{attribute 'GeneratedUsingTerminal: KL9940-0050'}
{attribute addProperty BoxType "KL9940-0050"}
{attribute addProperty Id "Channel_1AT %I*Channel_954C2EED0"}
{attribute addProperty CRC "782859838"}
{attribute addProperty Size "0"}
TYPE KL_2EA97E3E :
STRUCT
	{attribute addProperty Name "Channel_1"}
	Channel_1 : Channel_954C2EED;
END_STRUCT
END_TYPE

(* stored: Version 1.2.0.0, ProductVersion 3.1.4024.9
   DUT KL_2EA97E3E: Id {1a28a85f-5d97-40d9-974c-846fbb970fc1} *)
